FUNCTION_BLOCK StatusWidget
VAR_INPUT
	text  : STRING;
	color : StatusColor;
END_VAR
VAR_OUTPUT
END_VAR
VAR_IN_OUT
END_VAR
VAR
END_VAR

END_FUNCTION_BLOCK

(* stored: Version 1.1.0.1, ProductVersion 3.1.4018.2
   POU StatusWidget: Id {06bd82d5-1bda-49d6-920b-7e6bf7cb9442}, SpecialFunc None *)
